//{attribute 'qualified_only'}
VAR_GLOBAL
	E1 AT %I* : BOOL;
	S1 AT %Q* : BOOL;
END_VAR

(* stored: Version 1.1.0.1, ProductVersion 3.1.4024.12
   GVL GVL_Safety: Id {365b6964-9e64-42de-9533-3030fee7a8a9} *)
